INTERFACE I_Drive

{attribute 'monitoring':='call'}
PROPERTY Active : BOOL
GET
END_GET
END_PROPERTY

{attribute 'monitoring':='call'}
PROPERTY Error : BOOL
GET
END_GET
END_PROPERTY

METHOD reset : BOOL
VAR_INPUT
END_VAR
END_METHOD

METHOD ABSTRACT stop : BOOL
VAR_INPUT
END_VAR
END_METHOD

END_INTERFACE

(* stored: Version 1.1.0.1, ProductVersion 3.1.4024.11
   Itf I_Drive: Id {97843c9c-50ee-4368-8fd5-ec6e4d921ad0}
   Property Active: Id {22f2c010-e5b4-4e6f-ae07-528442546c4a}
   Get Get: Id {ac46d058-d832-4885-9e23-835c98ce5c95}
   Property Error: Id {b33f8b6d-756e-4d55-8410-5d769326987c}
   Get Get: Id {ad8d4ecb-7588-4940-a915-12e099739110}
   Method reset: Id {78774315-3cbe-4e9e-9d23-8faa39eac41e}
   Method stop: Id {8a7e512c-d54f-4452-a55b-3ee979f4c06a} *)
